# B&R Automation Studio project DO_Workshop
Automation Studio 

## Logical view

### Program Logical/Merge

#### Variables.var
```iecst
VAR
	Output1 : REAL;
	Input1 : REAL;
	var1 : REAL;
END_VAR
```

#### Merge.st
```iecst
PROGRAM _INIT

END_PROGRAM

PROGRAM _CYCLIC

	Output1		:= Input1;

	// TODO - Enter your line of code on the line below.  Perform math operations on Input1 and assign to Output1
<<<<<<< .merge_file_jWiUXq
	Output1		:= Input1 * 100.0 / 65.0;
=======

	Output1:= Input1 / var1;

>>>>>>> .merge_file_CMkzzj

END_PROGRAM

PROGRAM _EXIT
	(* Insert code here *)

END_PROGRAM
```

#### Merge_BACKUP_1851.st
```iecst
PROGRAM _INIT

END_PROGRAM

PROGRAM _CYCLIC

	Output1		:= Input1;

	// TODO - Enter your line of code on the line below.  Perform math operations on Input1 and assign to Output1
<<<<<<< HEAD
	Output1		:= Input1 * 100.0 / 65.0;
=======

	Output1:= Input1 / var1;

>>>>>>> develop

END_PROGRAM

PROGRAM _EXIT
	(* Insert code here *)

END_PROGRAM
```
